FUNCTION_BLOCK ArgQueue
VAR_GENERIC CONSTANT
	nCap		: UDINT := 100;
END_VAR

IMPLEMENTS I_MutArgQueue

VAR
	_list		: ArgList<nCap>;
	_nHead		: UDINT := 1;
	_nTail		: UDINT := 1;
END_VAR

PROPERTY Head : UDINT
GET
Head := _nHead;
END_GET
END_PROPERTY

PROPERTY List : I_ArgList
GET
List := _list;
END_GET
END_PROPERTY

METHOD Pop : Result
VAR_OUTPUT
	iArg	: I_Arg;
END_VAR
IF IsOk(_list.Get(_nTail, iArg => iArg), nOut => Pop) THEN
	_nTail := _nTail + 1;
	IF _nTail = nCap THEN
		_nTail := 1;
	END_IF
END_IF
END_METHOD

METHOD Push : Result
VAR_INPUT
	iArg		: I_Arg;
END_VAR
IF _nHead = _nTail THEN
	Push := Err.Ovf;
	RETURN;
END_IF

IF IsOk(_list.Append(iArg, _nHead), nOut => Push) THEN
	_nHead := _nHead + 1;
	IF _nHead = nCap THEN
		_nHead := 1;
	END_IF
END_IF
END_METHOD

PROPERTY Tail : UDINT
GET
Tail := _nTail;
END_GET
END_PROPERTY

END_FUNCTION_BLOCK

(* stored: Version 1.1.0.1
   POU ArgQueue: Id {5fefed48-7bae-45b6-a5e2-f3473e48d477}, SpecialFunc None
   Property Head: Id {212475c4-e8c8-4d1b-a3ee-53654d6c7959}
   Get Get: Id {a9358f8b-2ada-4118-b863-513c0b85c740}
   Property List: Id {7bb419a2-9a05-4640-9427-d39f30187a46}
   Get Get: Id {a822b4ee-ebcd-431d-bee5-1b2176157c94}
   Method Pop: Id {c0e476b5-0312-468c-bd79-2e025a1976a9}
   Method Push: Id {4cffbac1-66d4-4260-a313-b7e0e1c784cf}
   Property Tail: Id {0030fa0d-2cec-40bb-9189-8d4288b9442f}
   Get Get: Id {09bdafc1-07ce-41b5-9418-66d1d38d8e89} *)
